// TwinCAT 3 PLC project PLC3
// ProgramVersion: 3.1.4024.0
// libraries:
//   Tc2_MC2, * (Beckhoff Automation GmbH)
//   Tc2_Standard, * (Beckhoff Automation GmbH)
//   Tc2_System, * (Beckhoff Automation GmbH)
//   Tc3_Module, * (Beckhoff Automation GmbH)
//   Util, * (System)
// project tree:
//   / GlobalTextList.TcGTLO, Main_Visu.TcVIS, PlcTask.TcTTO, Task_2.TcTTO, 视图管理器.TcVMO (not stored)
//   GVLs/ GVL.TcGVL
//   POUs/ MAIN.TcPOU, PRG_LD.TcPOU
// real-time tasks:
//   TASK Task 1: cycle T#20ms, priority 20, ADS port 350
//   TASK Task 2: cycle T#4ms, priority 4, ADS port 351
//   TASK PlcTask: cycle T#10ms, priority 21, ADS port 352
// motion (NC):
//   TASK NC-Task 1 SAF: cycle T#1ms, priority 5, ADS port 501
//   TASK NC-Task 1 SVB: cycle T#4ms, priority 9, ADS port 511
//   AXIS Axis 1 (id 1)
//     Velo: SlowManual=360, FastManual=720, Maximum=888888
//     PositionAreaControl: Range=10
//     OtherSettings: AllowMotionCmdToSlave=true
//     encoder EncType=4
//       EncPara: ScaleFactorNumerator=1, ScaleFactorDenominator=16777216, Inverse=true, MaxCount=#x0000ffff
//         Inc: RefMode=2
//     drive DrvType=5
//       DrvPara: Inverse=true
//         Analog: VeloReferenz=888888, TorqueSetpointScale=10, ScaleFactorActTorque=0.1
//         TimeComp: TaskDelayCycles=1
//     controller CtrType=1
//       CtrPara: PriorControlFactor=1
//         PosDiffControl: Enable=false
//         PID: PosKp=5
//         Observer: BandWidth=20
//   AXIS Axis 2 (id 2)
//     Dynamic: Acceleration=93324, Deceleration=93324, Jerk=3266340
//     Velo: Maximum=6666
//     OtherSettings: AllowMotionCmdToSlave=true
//     encoder EncType=1
//     drive DrvType=5
//       Analog: TorqueSetpointScale=10, ScaleFactorActTorque=0.1
//     controller CtrType=1
//       CtrPara: PriorControlFactor=1
//         Observer: BandWidth=20
// I/O:
//   DEVICE Device 1 (EtherCAT), AmsNetId 192.168.199.183.2.1
//     Term 1 (EK1100) [EK1100 EtherCAT Coupler (2A E-Bus)]
//       Term 2 (EL2008) [EL2008 8Ch. Dig. Output 24V, 0.5A]
//       Term 3 (EL3174) [EL3174 4Ch. Ana. Input +/-10V Diff., +/-20mA SingleEnded, 16 Bit]
//     Drive 4 (AX5106-0000-0214) [AX5106-0000-0214 EtherCAT Drive (SoE, 1 Ch.)]
// variable links:
//   PLC3 Instance <-> NC-Task 1 SAF/Axes/Axis 1
//     Task_2 Inputs/GVL.Ax.NcToPlc <-> Outputs/ToPlc
//     Task_2 Outputs/GVL.Ax.PlcToNc <-> Inputs/FromPlc

CONFIGURATION PLC3
    RESOURCE PLC ON TwinCAT3
        TASK PlcTask(INTERVAL := T#10ms, PRIORITY := 21);
        TASK Task_2(INTERVAL := T#4ms, PRIORITY := 4);
        PROGRAM MAIN WITH PlcTask : MAIN;
        PROGRAM PRG_LD WITH Task_2 : PRG_LD;
    END_RESOURCE
END_CONFIGURATION

// ---- GVLs/GVL.TcGVL
{attribute 'qualified_only'}
VAR_GLOBAL
	Ax		:axis_ref;
END_VAR

// ---- POUs/MAIN.TcPOU
PROGRAM MAIN
VAR
	iTest		:INT;
	el2008	AT%Q*		:ARRAY[1..4] OF BOOL;
	fbBlink				:BLINK;
END_VAR

iTest := iTest + 1;

//fbBlink(ENABLE:=TRUE,TIMEHIGH:=T#500MS,TIMELOW:=T#500MS);
fbBlink(ENABLE:=TRUE,TIMEHIGH:=T#100MS,TIMELOW:=T#200MS);
el2008[2] := fbBlink.OUT;

END_PROGRAM

// ---- POUs/PRG_LD.TcPOU
PROGRAM PRG_LD
VAR
	MC_Power_0: MC_Power;
	MC_Jog_0: MC_Jog;
END_VAR

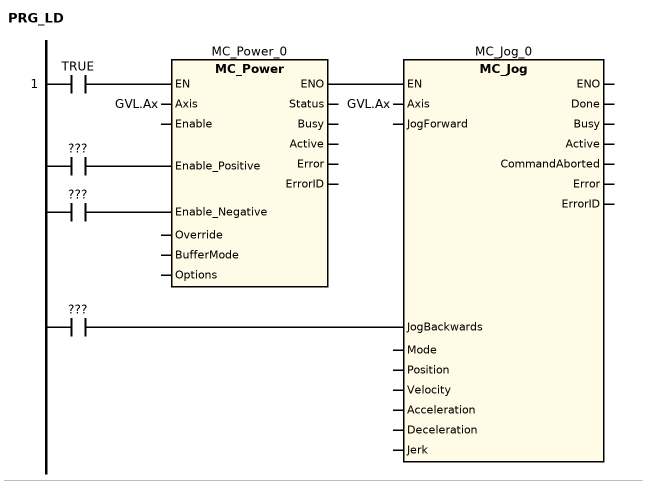
// NETWORK 1
MC_Power_0(Axis := GVL.Ax); // MC_Power
MC_Jog_0(Axis := GVL.Ax); // MC_Jog

END_PROGRAM

// ---- Main_Visu.TcVIS
VISUALIZATION Main_Visu  // 2x2
END_VISUALIZATION
